TYPE ST_P_RESET :
STRUCT
	Block:		INT;
	Channel:	ENUM_CHANNEL;
	ExecuteOnFail:	BOOL;
END_STRUCT
END_TYPE

(* stored: Version 1.1.0.1, ProductVersion 3.1.4024.10
   DUT ST_P_RESET: Id {5b34ddac-d5b5-40b0-9fd9-c5d81d9553e2} *)
